Universal Robots PolyScope program: 1_home_to_hover.urp

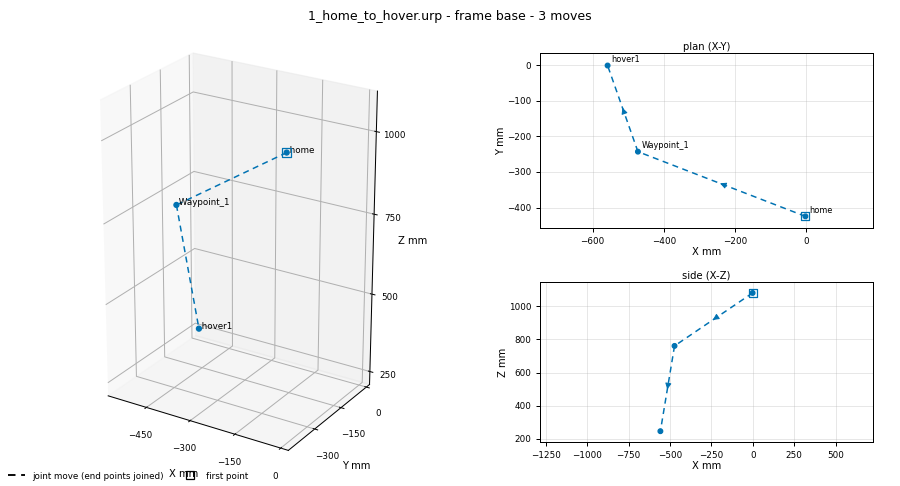
[picture p0: tool path of 1_home_to_hover.urp in frame base, 3 of 3 moves have a stored position in this frame; points joined in program order, loops and branches not executed]
Program 1_home_to_hover (installation=default directory=/programs/washer_rahman createdIn=5.9.5.1031259 lastSavedIn=5.9.5.1031259 robotSerialNumber=20215500597)
Calibrated DH parameters: a=[0.000193, -0.066673, -0.391568, -0.000012, 0.00005, 0]; d=[0.162643, -472.05677, 465.132521, 7.058239, 0.099746, 0.099582]; alpha=[1.571116, 0.00089, 0.003862, 1.569269, -1.569248, 0]; deltaTheta=[0, -1.413394, 7.628392, 0.068187, 0, -0.000001]
Robot Program (runOnlyOnce=true)
  MoveJ speed 60 deg/s, acceleration 80 deg/s^2 (useActiveTCP=true) feature=Base
    Waypoint home: TCP in base x=-1.584 y=-424.817 z=1080.554 mm, rx=-0.0045 ry=-2.2185 rz=2.2204 rad; joints [0, -89.999, 0.002, -90, -0.001, -0.001] deg; TCP offset x=0 y=0 z=191.5 mm, rx=0 ry=0 rz=0 rad
    MoveJ speed 60 deg/s, acceleration 80 deg/s^2 (useActiveTCP=true) feature=Base
      Waypoint Waypoint_1: TCP in base x=-472.633 y=-242.885 z=760.991 mm, rx=-0.4168 ry=-1.9658 rz=1.9427 rad; joints [-25.981, -98.486, 86.826, -170.504, -0.064, 0.002] deg
    URCap Gripper (Robotiq_Grippers, Robotiq Inc.) dataModel(position=0.0, force=100.0, speed=100.0, positionInDouble=0.0, forceInDouble=100.0, speedInDouble=100.0, slaveIds=[9], blocking=true)
  MoveJ speed 60 deg/s, acceleration 80 deg/s^2 (useActiveTCP=true) feature=Base
    Waypoint hover1: TCP in base x=-557.942 y=-0.628 z=246.464 mm, rx=-1.2338 ry=-1.2229 rz=1.2356 rad; joints [-31.234, -63.251, 147.705, -263.24, -57.851, 1.053] deg
  SuppressedNode
    MoveJ speed 60 deg/s, acceleration 80 deg/s^2 (useActiveTCP=true) feature=Base
      SuppressedNode
        Waypoint Waypoint (Variable): variable=glass_hover
